FUNCTION F_LogA1 
VAR_INPUT
	eLogLevel		: E_LogLevel;
	sLogger			: T_MaxString;
	sMessage		: T_MaxString;
	aArg1			: ANY;
END_VAR

F_LogLA1(eLogLevel, Const.sGlobalLogger, sMessage, aArg1);

END_FUNCTION

(* stored: Version 1.1.0.1, ProductVersion 3.1.4024.0
   POU F_LogA1: Id {fbb41f90-470a-440a-900e-95d2040a9b4c}, SpecialFunc None *)
